INTERFACE IProcess

PROPERTY EndPosition : MC_LREAL
GET
END_GET
END_PROPERTY

PROPERTY ProcessVelocity : mc_lreal
GET
END_GET
END_PROPERTY

END_INTERFACE

(* stored: Version 1.1.0.1
   Itf IProcess: Id {35f38492-ddb4-43cb-90ed-57490b1c2a0f}
   Property EndPosition: Id {dd6f2210-a4af-4fbc-a10a-6e02b45480ee}
   Get Get: Id {31f9cf28-dd57-4d20-ace6-7cac7fc9bf57}
   Property ProcessVelocity: Id {4148105b-d9b1-443c-b3c0-196030eb7c2f}
   Get Get: Id {4f40390c-f906-437a-882e-04f737dbad29} *)
